FUNCTION_BLOCK FB_MonetTelescopeControl EXTENDS FB_AltAzTelescopeControl IMPLEMENTS I_AltAzTelescope
VAR_INPUT
	fbFocus				: I_Focus;
	fbCovers			: I_MirrorCovers;
	fbBrake				: I_Brake;	
	fbHydraulics   		: I_Hydraulics;
	fbElevation			: REFERENCE TO FB_ElevationControl;
	fbAzimuth			: REFERENCE TO FB_AzimuthControl;
	fbDerotator			: REFERENCE TO FB_DerotatorControl;

	bBrakeClearing		: BOOL	:= TRUE;
END_VAR
VAR_OUTPUT
	fDerotatorSign		: LREAL := 1.0;	// derotator
	
	fElevationPointingOffset : LREAL;
	fAzimuthPointingOffset : LREAL;
	fElevationPointingOffset2 : LREAL;
	fAzimuthPointingOffset2 : LREAL;
	
	fRightAscensionCurrentSky: LREAL;
	fDeclinationCurrentSky: LREAL;

	fDerotatorVelocity	: LREAL;	// rotational velocity of the derotator
	fElevationVelocity	: LREAL;	// rotational velocity of the elevation
	fAzimuthVelocity	: LREAL;	// rotational velocity of the elevation
END_VAR
VAR
	fbPointing			: FB_PointingModelForward(AOFF := 0.0, BNP := 0.0, AN_A := 0.0, AE_A := 0.0, NPAE := 0.0, 
                                                  EOFF := 0.0, AN_E := 0.0, AE_E := 0.0, TF := 0.0);
	fbPointingInverse	: FB_PointingModelInversion(fbPointing := fbPointing);
END_VAR

// get the system time
fbTime();
fJd := DateTime2JD(fbTime.time_RTCEX2);
fLst := CT2LST(telescopeConfig.longitude, fJd);

// set reset state either by hardware (key pressed) or by software (set by e.g. tcs)
rtrigReset(CLK := bReset);

IF bReset THEN
	bHorizonError := FALSE; // if reset, the bHorizonError can be switched off
	
	// reset the stages of all statemachine methods
	bInterrupted := TRUE; 
	_HomeTelescope();
	_GotoTelescope();
	_SlewTelescope();
	_ParkTelescope();
	bInterrupted := FALSE;
END_IF

// get error ID, reset if bReset command is set
IF fbAzimuth.Error THEN
	nErrorID := fbAzimuth.nErrorID;
	IF bReset THEN
		fbAzimuth.Reset();
	END_IF
ELSIF fbElevation.bError THEN
	nErrorID := fbElevation.nErrorID;
	IF bReset THEN
		fbElevation.Reset();
	END_IF
ELSIF fbDerotator.bError THEN
	nErrorID := fbDerotator.nErrorID;
	IF bReset THEN
		fbDerotator.Reset();
	END_IF	
ELSIF fbFocus <> 0 AND_THEN fbFocus.Error THEN
	nErrorID := fbFocus.ErrorID;
	IF bReset THEN
		fbFocus.Reset();
	END_IF
END_IF

// fSlewTime
fSlewTime :=  MAX(MAX(fbElevation.fSlewTime, fbAzimuth.fSlewTime), fbDerotator.fSlewTime);

bError := fbElevation.Error OR 
		 fbAzimuth.bError OR
		 (fbFocus <> 0 AND_THEN fbFocus.Error) OR
		 fbDerotator.bError;
			
IF bError THEN
	bGoHome := 	FALSE;
	bTrack := 	FALSE;
	bGoto := 	FALSE;
	bSlew := 	FALSE;
	fbElevation.Enable := FALSE;
	fbAzimuth.Enable := FALSE;
	fbDerotator.Enable := FALSE;
ELSE
	nErrorID := 0;
END_IF

IF fbElevation.bError THEN
	fbElevation.Enable := FALSE;
	fbAzimuth.Enable := FALSE;
	fbDerotator.Enable := FALSE;
	fbBrake.CloseBrake();
END_IF

eq2hor(
	ra := fRightAscension,
	dec := fDeclination,
	lon := telescopeConfig.longitude,
	lat := telescopeConfig.latitude,
	altitude := telescopeConfig.altitude,
	JD := fJd + fTimeOffset,
	refract_to_observed := TRUE,
	// refract := FALSE,
	alt => fElevationCalc,
	az => fAzimuthCalc,
	ha => fHourAngleCalc);

// apply pointing model
fbPointing(
	fAzimuth			:= fAzimuthCalc,
	fElevation			:= fElevationCalc,
	fAzimuthOffset		=> fAzimuthPointingOffset,
	fElevationOffset	=> fElevationPointingOffset
);
fElevationCalc := fElevationCalc + fElevationPointingOffset + fElevationOffset;
fAzimuthCalc := fAzimuthCalc + fAzimuthPointingOffset + fAzimuthOffset / COS(fElevationCalc * d2r);

// calculate derotator position 
fDerotatorCalc := F_DerotatorPosition2(fAzimuthCalc, fElevationCalc, fDeclination, telescopeConfig.latitude, fDerotatorSign)  + fDerotatorOffset;

// calculate velocities
fDerotatorVelocity := F_Derotatorvelocity(fElevationCalc, fAzimuthCalc, telescopeConfig.latitude);
fElevationVelocity := F_Elevationvelocity(fAzimuthCalc, telescopeConfig.latitude);
fAzimuthVelocity := F_Azimuthvelocity(fElevationCalc, fAzimuthCalc, telescopeConfig.latitude);

// calculate velocities
fDerotatorVelocity := F_Derotatorvelocity(fElevationCalc, fAzimuthCalc, telescopeConfig.latitude);
fElevationVelocity := F_Elevationvelocity(fAzimuthCalc, telescopeConfig.latitude);
fAzimuthVelocity := F_Azimuthvelocity(fElevationCalc, fAzimuthCalc, telescopeConfig.latitude);

IF (fAzimuthCalc > 270.0) THEN
	fAzimuthCalc := fAzimuthCalc - 360.0;
ELSIF (fAzimuthCalc < -274.0) THEN
	fAzimuthCalc := fAzimuthCalc + 360.0;
END_IF
IF (fDerotatorCalc > 360.0) THEN
	fDerotatorCalc := fDerotatorCalc - 360.0;
ELSIF (fDerotatorCalc < -90.0) THEN
	fDerotatorCalc := fDerotatorCalc + 360.0;
END_IF

//IF (fAzimuthCalc > 310.0 AND fAzimuthVelocity > 0.0) OR (fAzimuthCalc > 440.0) THEN
//	fAzimuthCalc := fAzimuthCalc - 360.0;
//ELSIF (fAzimuthCalc < 80.0 AND fAzimuthVelocity < 0.0) OR (fAzimuthCalc < -50.0) THEN
//	fAzimuthCalc := fAzimuthCalc + 360.0;
//END_IF

//IF (fDerotatorCalc > 290.0 AND fDerotatorVelocity > 0.0) OR (fDerotatorCalc > 380.0) THEN
//	fDerotatorCalc := fDerotatorCalc - 360.0;
//ELSIF (fDerotatorCalc < 20.0 AND fDerotatorVelocity < 0.0) OR (fDerotatorCalc < -70.0) THEN
//	fDerotatorCalc := fDerotatorCalc + 360.0;
//END_IF

// get current coordinates	
fAzimuthCurrent := fbAzimuth.fActualPosition;
fElevationCurrent := fbElevation.fActualPosition;
fDerotatorCurrent := fbDerotator.fActualPosition;

// apply inverse pointing model
fbPointingInverse(
	fAzimuth			:= fAzimuthCurrent,
	fElevation			:= fElevationCurrent,
	fAzimuthOffset  	=> fAzimuthPointingOffset2,
	fElevationOffset	=> fElevationPointingOffset2
);
fAzimuthCurrentSky := fAzimuthCurrent - fAzimuthPointingOffset2;
fElevationCurrentSky := fElevationCurrent - fElevationPointingOffset2;

// add offsets
//fElevationCurrent := fElevationCurrentSky - fElevationOffset;
//fAzimuthCurrent := fAzimuthCurrentSky - fAzimuthOffset / COS(fElevationCalc * d2r);

// calculate equatorial coordinates
hor2eq(alt := fElevationCurrentSky - fElevationOffset, 
		az := fAzimuthCurrentSky - fAzimuthOffset / COS(fElevationCalc * d2r),
		jd := fJd,
		lat := telescopeConfig.latitude,
		lon := telescopeConfig.longitude,
		altitude := telescopeConfig.altitude,
		refract_to_observed := FALSE,
		// refract := FALSE,
		ra => fRightAscensionCurrent,
		dec => fDeclinationCurrent);		
hor2eq(alt := fElevationCurrentSky, 
		az := fAzimuthCurrentSky,
		jd := fJd,
		lat := telescopeConfig.latitude,
		lon := telescopeConfig.longitude,
		altitude := telescopeConfig.altitude,
		refract_to_observed := FALSE,
		ra => fRightAscensionCurrentSky,
		dec => fDeclinationCurrentSky);
	
// If the Telescope dips under the fHorizon (e.g. while tracking, stop and gohome)
IF fbElevation.Calibrated AND fElevationCurrent < (fHorizon+0.2) THEN
	IF NOT bStopped AND NOT bGoHome THEN
		bStop := TRUE;
	ELSE
		bGoHome := TRUE;
	END_IF
END_IF
		
tpPowerOnWarning(IN := bPower OR (NOT fbElevation.bEnable AND fbBrake.BrakeOpen), PT := T#250MS);

tonPowerTimeout(IN := TCS_command = E_TCSCommand.no_command AND NOT bIsParked, PT := T#12H);
tonCommandTimeout();
IF tonPowerTimeout.Q AND NOT bIsParked THEN
	bPark := TRUE;
END_IF
		
// set TCS_command according to state variables ordered by precedence
IF bPower THEN
	TCS_command := E_TCSCommand.poweron;
	
ELSIF bStop THEN
	bTrack := FALSE;
	
	// If the stop is during a movement, reset the stage of the movement first
	IF bPark THEN
		bPark := FALSE;
		_ParkTelescope();
	ELSIF bGoto THEN
		bGoto := FALSE;
		_GotoTelescope();
	ELSIF bSlew THEN
		bSlew := FALSE;
		_SlewTelescope();
	ELSIF bGoHome THEN
		bGoHome := FALSE;
		_HomeTelescope();
	END_IF
	TCS_command := E_TCSCommand.stop;
	
ELSIF bPark THEN
	bTrack := FALSE;
	// If lower presedence commands are ongoing, let them know they are interupted
	IF bGoto OR bSlew OR bGoHome THEN
		bGoHome := FALSE;
		bGoto := FALSE;
		bSlew := FALSE;
		bInterrupted := TRUE;
		_HomeTelescope();
		_GotoTelescope();
		_SlewTelescope();
		
	ELSE
		IF bReady AND NOT bBusy THEN
			bInterrupted := FALSE;
			TCS_command := E_TCSCommand.park;
		END_IF
	END_IF
	
ELSIF bGoHome THEN
	bTrack := FALSE;
	// If lower presedence commands are ongoing, let them know they are interupted
	IF bGoto OR bSlew THEN
		bGoto := FALSE;
		bSlew := FALSE;
		bInterrupted := TRUE;
		_GotoTelescope();
		_SlewTelescope();
		
	ELSE
		IF bReady AND NOT bBusy AND bStopped THEN
			bInterrupted := FALSE;
			TCS_command := E_TCSCommand.gohome;
		END_IF
	END_IF
	
	
ELSIF bGoto THEN
	bTrack := FALSE;
	// If lower presedence commands are ongoing, let them know they are interupted
	IF bSlew THEN
		bSlew := FALSE;
		bInterrupted := TRUE;
		_SlewTelescope();
	ELSE
		IF bReady AND NOT bBusy THEN
			bInterrupted := FALSE;
			TCS_command := E_TCSCommand.goto;
		END_IF
	END_IF
		
ELSIF bSlew THEN
	bTrack := FALSE;
	IF bReady AND NOT bBusy THEN
		TCS_command := E_TCSCommand.slew;
	END_IF
	
ELSIF bTrack THEN
	IF bReady AND NOT bBusy THEN
		TCS_command := E_TCSCommand.track;
	END_IF
	
ELSE
	TCS_command := E_TCSCommand.no_command;
	fbElevation.bMoveAxis := FALSE;
	fbAzimuth.bMoveAxis := FALSE;
	fbDerotator.bMoveAxis := FALSE;
	fbElevation.bTracking := FALSE;
	fbAzimuth.bTracking := FALSE;
	fbDerotator.bTracking := FALSE;
END_IF

IF TCS_command = E_TCSCommand.poweron THEN
	_PowerOn();
	tonCommandTimeout(IN := TCS_command = E_TCSCommand.poweron, PT := T#12H);
	TCSCTOEvent.OnMessage := 'POWER';
ELSIF TCS_command = E_TCSCommand.stop THEN
	_StopTelescope();
	tonCommandTimeout(IN := TCS_command = E_TCSCommand.stop, PT := T#2S);
	TCSCTOEvent.OnMessage := 'STOP';
ELSIF TCS_command = E_TCSCommand.park THEN
	_ParkTelescope();
	tonCommandTimeout(IN := TCS_command = E_TCSCommand.park, PT := T#2M);
	TCSCTOEvent.OnMessage := 'PARK';
ELSIF TCS_command = E_TCSCommand.gohome THEN
	_HomeTelescope();
	tonCommandTimeout(IN := TCS_command = E_TCSCommand.gohome, PT := T#2M);
	TCSCTOEvent.OnMessage := 'GOHOME';
ELSIF TCS_command = E_TCSCommand.goto THEN
	_GotoTelescope();
	tonCommandTimeout(IN := TCS_command = E_TCSCommand.goto, PT := T#2M);
	TCSCTOEvent.OnMessage := 'GOTO';
ELSIF TCS_command = E_TCSCommand.slew THEN
	_SlewTelescope();
	tonCommandTimeout(IN := TCS_command = E_TCSCommand.slew, PT := T#2M);
	TCSCTOEvent.OnMessage := 'SLEW';
ELSIF TCS_command = E_TCSCommand.track THEN
	_TrackTelescope();
	tonCommandTimeout(IN := TCS_command = E_TCSCommand.track, PT := T#12H);
	TCSCTOEvent.OnMessage := 'TRACK';
ELSE
	// disable command timeout
	tonCommandTimeout(IN := FALSE);
	TCSCTOEvent.OnMessage := 'NOCOMMAND';
END_IF
 
bSlewing := NOT bTracking AND (fbElevation.fbAxis.InMotion OR fbElevation.fbAxis.InRamp OR
			fbAzimuth.fbAxis.InMotion OR fbAzimuth.fbAxis.InRamp OR
			fbDerotator.fbAxis.InMotion OR fbDerotator.fbAxis.InRamp);

// signal must be stable for 5500MS
tonTrackingDelay(in := fbElevation.fbAxis.isTracking AND 
			fbAzimuth.fbAxis.isTracking AND
			fbDerotator.fbAxis.isTracking,PT :=T#5500MS, Q => bTracking);
			
bStopped :=  (NOT fbElevation.bEnable OR fbElevation.fbAxis.StandStill) AND 
			(NOT fbAzimuth.bEnable OR fbAzimuth.fbAxis.StandStill) AND
			(NOT fbDerotator.bEnable OR fbDerotator.fbAxis.StandStill);
			
bHomed := fbElevation.Calibrated AND
			fbAzimuth.Calibrated AND
			fbFocus.Calibrated AND
			fbDerotator.Calibrated;
			
bReady := bHomed AND 
	fbCovers.Opened AND 
	fbElevation.bEnable AND
	fbAzimuth.bEnable AND
	fbDerotator.bEnable AND fbBrake.BrakeOpen AND 
    NOT bError;

bBusy := fbElevation.fbAxis.Busy OR
		fbAzimuth.fbAxis.Busy OR
		fbDerotator.fbAxis.Busy OR
		fbFocus.Busy;

(* STATUS STATES*)
//fReadyState (see also _PowerOn and _ParkTelescope calls above)
IF bReady THEN
	fReadyState := 1.0;
ELSIF bError THEN
	fReadyState := -1.0;
ELSIF bPower THEN
	fReadyState := 0.7;
ELSIF bIsParked THEN
	fReadyState := 0.0;
ELSIF bPark THEN
	fReadyState := 0.3;
END_IF

//MotionState
IF bStopped THEN
	nMotionState := 0;
ELSIF bSlewing OR bBusy THEN
	nMotionState := 1;
ELSIF bTracking THEN
	nMotionState := 8;
END_IF

// unset the STOP command if telescope is already stopped
IF bStopped THEN
	bStop := FALSE;
END_IF
	
IF NOT bError THEN
	bReset := FALSE;
END_IF

IF bEstopTriggered THEN
	fbElevation.Enable := FALSE;
	fbAzimuth.Enable := FALSE;
	fbDerotator.Enable := FALSE;
END_IF

// send telemetry
IF bSlewing OR bTrack OR bTracking THEN
	tonMQTTTimer.PT := T#500MS; // during movement every second
ELSE
	tonMQTTTimer.PT := T#1000MS; // otherwise every five seconds
END_IF
tonMQTTTimer(IN:=TRUE);
IF tonMQTTTimer.Q THEN
	tonMQTTTimer(IN:=FALSE);
	_SendTelemetry();
END_IF


(* Event function blocks start here. *)
TCSpowerEvent(	Trigger := bPowerFailure, 
				Level := ADSLOG_MSGTYPE_ERROR,
				FormatString := 'power %s',
				//OnMessage := 'Failure',
				OffMessage := 'OK', 
				Comm := fbComm);

TCSgohomeEvent(	Trigger := bGoHome, 
				Level := ADSLOG_MSGTYPE_HINT,
				FormatString := 'GOHOME %s',
				OnMessage := 'commencing',
				OffMEssage := 'completed', 
				Comm := fbComm);
TCSparkEvent(	Trigger := bPark, 
				Level := ADSLOG_MSGTYPE_HINT,
				FormatString := 'PARK %s',
				OnMessage := 'commencing',
				OffMEssage := 'completed', 
				Comm := fbComm);
TCSgotoEvent(	Trigger := bGoto, 
				Level := ADSLOG_MSGTYPE_HINT,
				FormatString := 'GOTO %s',
				OnMessage := 'commencing',
				OffMEssage := 'completed', 
				Comm := fbComm);
TCStrackEvent(	Trigger := bTrack, 
				Level := ADSLOG_MSGTYPE_HINT,
				FormatString := 'TRACK %s',
				OnMessage := 'commencing',
				OffMEssage := 'completed', 
				Comm := fbComm);
TCSstopEvent(	Trigger := bStop, 
				Level := ADSLOG_MSGTYPE_WARN,
				FormatString := 'STOP %s',
				OnMessage := 'commencing',
				OffMEssage := 'completed',
				OffLevel := ADSLOG_MSGTYPE_HINT, 
				Comm := fbComm);
TCStargetHorizonEvent(	Trigger := bPower AND fElevationCalc<fHorizon, 
				Level := ADSLOG_MSGTYPE_WARN,
				FormatString := '%s',
				OnMessage := 'Target below safe horizon',
				OffMEssage := '', 
				Comm := fbComm);
TCSreadyEvent(	Trigger := bPower AND bReady, 
				Level := ADSLOG_MSGTYPE_HINT,
				FormatString := '%s',
				OnMessage := 'STELLA1 startup finished', 
				Comm := fbComm);
TCSCTOEvent(	Trigger := tonCommandTimeout.Q,
				Level := ADSLOG_MSGTYPE_WARN,
				FormatString := 'A timeout occured during %s command!',
				OnMessage := 'NOCOMMAND', 
				Comm := fbComm);

METHOD PRIVATE _GotoTelescope : USINT
VAR_INPUT
END_VAR
VAR
	GoToEvent		: FB_Eventlog;
	commandTimeout	: TON;
END_VAR
VAR_STAT
	nStage			: USINT := 0;
	nLastStage		: USINT := 101;
END_VAR
_GotoTelescope := nStage;
commandTimeout(IN := nStage < 100, PT := T#600S);
IF commandTimeout.Q THEN
	bError := TRUE;
	nErrorID := 16#10;
	bGoto := FALSE;
	nStage := 0;
	RETURN;
END_IF

IF fElevationCalc<2.0 THEN
	bError := TRUE;
	nErrorID := 16#15;
	bGoto := FALSE;
	nStage := 0;
	RETURN;
END_IF

IF bReset OR bError OR bInterrupted THEN
	nStage := 0;
	RETURN;
END_IF

CASE nStage OF
	0:	
		IF bReady AND NOT bBusy THEN
			nStage := 10;
		END_IF
	10:
		IF fbElevation.Tracking = TRUE OR fbAzimuth.Tracking = TRUE OR fbDerotator.Tracking = TRUE THEN
			fbElevation.Tracking := FALSE;
			fbAzimuth.Tracking := FALSE;
			fbDerotator.Tracking := FALSE;
		ELSE
			nStage := 25;
		END_IF				
	25:	
		fbElevation.Position := fElevationCalc;
		fbAzimuth.Position := fAzimuthCalc;
		fbDerotator.Position := fDerotatorCalc;
		fbDerotator.Velocity := 10.0;
		fbElevation.Velocity := 10.0;
		fbAzimuth.Velocity := 10.0;
		
		fbElevation.MoveAxis := TRUE;
		fbAzimuth.MoveAxis := TRUE;
		fbDerotator.MoveAxis := TRUE;
		IF fbElevation.Busy AND
			fbAzimuth.Busy AND
			fbDerotator.Busy THEN
				nStage := 50;
		END_IF
	50:
		IF NOT fbElevation.Busy AND fbElevation.MoveDone THEN
			fbElevation.MoveAxis := FALSE;
		END_IF
		IF NOT fbAzimuth.Busy AND fbAzimuth.MoveDone THEN
			fbAzimuth.MoveAxis := FALSE;
		END_IF
		IF NOT fbDerotator.Busy AND fbDerotator.MoveDone THEN
			fbDerotator.MoveAxis := FALSE;
		END_IF
		IF NOT fbElevation.MoveAxis AND 
           NOT fbAzimuth.MoveAxis AND 
		   NOT fbDerotator.MoveAxis THEN
		   nStage := 75;
		END_IF
	75:
		IF NOT bSlewing AND bStopped THEN // all axis standstill
			nStage := 100;
		END_IF
	100:
		fbElevation.MoveAxis := FALSE;
		fbAzimuth.MoveAxis := FALSE;
		fbDerotator.MoveAxis := FALSE;
		fAzimuth := fAzimuthCalc;
		fElevation := fElevationCalc;
		bGoto := FALSE;
		// enable automatic tracking
		bTrack := bAutoTrack;
		nStage := 0;
END_CASE
GoToEvent(Trigger := nStage > nLastStage, FormatString := 'GoTo progress: %s', OnMessage := USINT_TO_STRING(nStage), comm := fbComm);
nLastStage := nStage;
END_METHOD

METHOD PRIVATE _HomeTelescope : BOOL
VAR_INPUT
END_VAR
VAR
	HomeEvent		: FB_Eventlog;
	commandTimeout	: TON;
END_VAR
commandTimeout(IN := NOT _HomeTelescope, PT := T#600S);
IF commandTimeout.Q THEN
	bError := TRUE;
	nErrorID := 16#30;
	_HomeTelescope :=TRUE;
END_IF

IF bReady AND bStopped AND NOT bBusy AND NOT bTracking THEN
	fbElevation.Velocity := 10.0;
	fbElevation.Position := telescopeConfig.elevationHome;
	fbElevation.MoveAxis := TRUE;
	fbAzimuth.Velocity := 10.0;
	fbAzimuth.Position := telescopeConfig.azimuthHome;
	fbAzimuth.MoveAxis := TRUE;
	fbDerotator.Velocity := 10.0;
	fbDerotator.Position := telescopeConfig.derotatorHome;
	fbDerotator.MoveAxis := TRUE;	
END_IF

IF fbElevation.MoveDone AND 
	fbAzimuth.MoveDone AND 
	fbDerotator.MoveDone THEN
	bGoHome := FALSE;
	fElevation := fElevationCurrent;
	fAzimuth := fAzimuthCurrent;
	_HomeTelescope := TRUE;
ELSE
	_HomeTelescope := FALSE;
END_IF

HomeEvent(Trigger := _HomeTelescope, 
			Level := ADSLOG_MSGTYPE_HINT,
			FormatString := '%s',
			OnMessage := 'Telescope is homed.', comm := fbComm);
END_METHOD

METHOD PRIVATE _ParkTelescope : USINT
VAR_INPUT
END_VAR
VAR
	ParkEvent	: FB_Eventlog;
END_VAR
VAR_STAT
	nStage		: USINT := 0;
	nLastStage	: USINT := 101;
END_VAR
_ParkTelescope := nStage;
IF bReset OR bError OR bStop OR bInterrupted THEN
	nStage := 0;
	RETURN;
END_IF
IF bIsParked THEN
	nStage := 100;
END_IF
CASE nStage OF
	0: 
		bGoHome := 	FALSE;
		bTrack := 	FALSE;
		bGoto := 	FALSE;
		bSlew := 	FALSE;
		IF fbFocus <> 0 THEN
			fbFocus.Position := telescopeConfig.focusPark;
		END_IF
		IF bError THEN // emergency park
			fbBrake.CloseBrake();
			fbElevation.Enable := FALSE;
			fbAzimuth.Enable := FALSE;
			fbDerotator.Enable := FALSE;	
			fbCovers.Close();	
			nStage := 80;
		END_IF
		nStage := 10;
	10:
		IF fbElevation.Tracking = TRUE OR fbAzimuth.Tracking = TRUE OR fbDerotator.Tracking = TRUE THEN
			fbElevation.Tracking := FALSE;
			fbAzimuth.Tracking := FALSE;
			fbDerotator.Tracking := FALSE;
		ELSE
			nStage := 20;
		END_IF		
	20:
		fbElevation.Position := telescopeConfig.elevationPark;
		fbElevation.Velocity := 10.0;
		fbElevation.MoveAxis := TRUE;
		fbAzimuth.Position := telescopeConfig.azimuthPark;
		fbAzimuth.Velocity := 10;
		fbAzimuth.MoveAxis := TRUE;
		fbDerotator.Position := telescopeConfig.derotatorPark;
		fbDerotator.Velocity := 10.0;
		fbDerotator.MoveAxis := TRUE;
		IF fbElevation.Busy AND
			fbAzimuth.Busy AND
			fbDerotator.Busy THEN
				nStage := 40;
		END_IF
	40:
		IF fbElevation.MoveDone THEN
			fbElevation.MoveAxis := FALSE;
		END_IF
		IF fbAzimuth.MoveDone THEN
			fbAzimuth.MoveAxis := FALSE;
		END_IF
		IF fbDerotator.MoveDone THEN
			fbDerotator.MoveAxis := FALSE;
		END_IF
		IF NOT bSlewing THEN // all axis standstill
			nStage := 60;
		END_IF
	60:
		IF NOT fbElevation.Enable AND NOT fbAzimuth.Enable AND NOT fbDerotator.Enable THEN
			nStage := 80;
		END_IF

		IF bStopped THEN
			fbElevation.Enable := FALSE;
			fbAzimuth.Enable := FALSE;
			fbDerotator.Enable := FALSE;
		END_IF
		
		fbElevation.bMoveAxis := FALSE;
		fbAzimuth.bMoveAxis := FALSE;
		fbDerotator.bMoveAxis := FALSE;
	80:
		IF fbElevation.Enable OR fbAzimuth.Enable OR fbDerotator.Enable THEN
			nStage := 60;
		END_IF
		IF NOT fbBrake.BrakeOpen THEN
			fbCovers.Close();
			fbHydraulics.Enable := FALSE;
		END_IF
		IF fbCovers.Closed THEN
			nStage := 100;
		END_IF
	100:
			bIsParked := TRUE;
			bPark := FALSE;
			_ParkTelescope := 100;
			nStage := 0;	
END_CASE
ParkEvent(Trigger := nStage > nLastStage, FormatString := 'Parking progress: %s', OnMessage := USINT_TO_STRING(nStage), comm := fbComm);
nLastStage := nStage;
END_METHOD

METHOD PRIVATE _PowerOn : BOOL
VAR_INPUT
END_VAR
IF NOT bBrakeClearing THEN
	bPowerFailure := TRUE;
	TCSpowerEvent.OnMessage := 'failure: brake clearing not set';
	bPower := FALSE;
ELSIF bError THEN
	bPowerFailure := TRUE;
	TCSpowerEvent.OnMessage := 'Generic error during power on occured.';
	bPower := FALSE;
ELSE
	bPowerFailure := FALSE;		
END_IF
// COVER MUST BE OPENED FOR A SUCCESSFUL WAKE & SHAKE COMMAND!
fbCovers.Open();

// enable elevation, enable azimuth
IF bMainReady AND fbCovers.Opened THEN
	fbElevation.Enable := TRUE;
	fbAzimuth.Enable := TRUE;
	fbDerotator.Enable := TRUE;
END_IF

IF fbElevation.Ready AND NOT fbElevation.Calibrated THEN
	fbElevation.HomeAxis := TRUE;
END_IF

IF fbAzimuth.Ready AND NOT fbAzimuth.Calibrated THEN
	fbAzimuth.HomeAxis := TRUE;
END_IF

// enable derotator
IF fbElevation.Ready THEN
	fbDerotator.HomeAxis := fbDerotator.Ready AND NOT fbDerotator.Calibrated;
END_IF

// start calibration of focus after elevation has been calibrated
// this avoids imbalance by the M2 mirror on the elvation during its calibration
IF fbElevation.Calibrated AND (fbFocus <> 0 AND_THEN NOT fbFocus.Calibrated) THEN
	fbFocus.Enable := TRUE;
	fbFocus.HomeAxis := TRUE;
END_IF

IF fbCovers.Opened AND 
	fbElevation.Calibrated AND
	fbAzimuth.Calibrated AND
	fbDerotator.Calibrated THEN
	//FocusControl.Calibrated THEN
	bPower := FALSE;
	_PowerOn := TRUE;
	bIsParked := FALSE;
	// slew the telescope to the home position
	bGoHome := TRUE;
ELSE
	_PowerOn := FALSE;
END_IF
END_METHOD

METHOD _SendTelemetry : BOOL
VAR_INPUT
END_VAR
SUPER^._PublishTelemetry();

fbComm.Publish('telescope', 'dome', 'TELESCOPE.READY_STATE',	LREAL_TO_STRING(fReadyState));
fbComm.Publish('telescope', 'dome', 'TELESCOPE.MOTION_STATE',	LREAL_TO_STRING(nMotionState));

// INFO
fbComm.Publish('telescope', 'dome', 'TELESCOPE.INFO.NAME',	telescopeConfig.name);
fbComm.Publish('telescope', 'dome', 'TELESCOPE.INFO.DIAMETER',	LREAL_TO_STRING(telescopeConfig.diameter));
fbComm.Publish('telescope', 'dome', 'TELESCOPE.INFO.CABINET',	telescopeConfig.cabinet);
fbComm.Publish('telescope', 'dome', 'TELESCOPE.INFO.MANUFACTURER', telescopeConfig.manufacturer);

// config
fbComm.Publish('telescope', 'dome', 'TELESCOPE.CONFIG.MOUNTOPTIONS', telescopeConfig.mountOptions);
fbComm.Publish('telescope', 'dome', 'TELESCOPE.CONFIG.MOUNT', telescopeConfig.mount);

// STATUS
IF bEstopTriggered THEN
	fbComm.Publish('telescope', 'dome', 'TELESCOPE.STATUS.GLOBAL', '1');
ELSIF bError THEN
	fbComm.Publish('telescope', 'dome', 'TELESCOPE.STATUS.GLOBAL', '2');
ELSE
	fbComm.Publish('telescope', 'dome', 'TELESCOPE.STATUS.GLOBAL', '0');
END_IF

// INSTRUMENTAL
fbComm.Publish('telescope', 'dome', 'OBJECT.INSTRUMENTAL.ALT', LREAL_TO_STRING(fElevation));
fbComm.Publish('telescope', 'dome', 'OBJECT.INSTRUMENTAL.AZ', LREAL_TO_STRING(fAzimuth));

// EQUATORIAL
fbComm.Publish('telescope', 'dome', 'OBJECT.EQUATORIAL.EPOCH', 'J2000.0');
fbComm.Publish('telescope', 'dome', 'OBJECT.EQUATORIAL.EQUINOX', 'J2000.0');
fbComm.Publish('telescope', 'dome', 'OBJECT.EQUATORIAL.RA_PM', '0.0');
fbComm.Publish('telescope', 'dome', 'OBJECT.EQUATORIAL.DEC_PM', '0.0');
fbComm.Publish('telescope', 'dome', 'OBJECT.EQUATORIAL.RA_RATE', '0.0');
fbComm.Publish('telescope', 'dome', 'OBJECT.EQUATORIAL.DEC_RATE', '0.0');
fbComm.Publish('telescope', 'dome', 'OBJECT.EQUATORIAL.RA', LREAL_TO_STRING(fRightAscension/15.0));
fbComm.Publish('telescope', 'dome', 'OBJECT.EQUATORIAL.DEC', LREAL_TO_STRING(fDeclination));	

// HORIZONTAL
fbComm.Publish('telescope', 'dome', 'OBJECT.HORIZONTAL.ALT', LREAL_TO_STRING(fElevationCalc));
fbComm.Publish('telescope', 'dome', 'OBJECT.HORIZONTAL.AZ', LREAL_TO_STRING(fAzimuthCalc));

(* POINTING *)
fbComm.Publish('telescope', 'dome', 'POINTING.SLEWTIME', LREAL_TO_STRING(fSlewtime));
fbComm.Publish('telescope', 'dome', 'POINTING.OFFSETS.ALT', LREAL_TO_STRING(fElevationPointingOffset));
fbComm.Publish('telescope', 'dome', 'POINTING.OFFSETS.AZ', LREAL_TO_STRING(fAzimuthPointingOffset));

(*POSITION*)
//LOCAL
fbComm.Publish('telescope', 'dome', 'POSITION.LOCAL.SIDEREAL_TIME', LREAL_TO_STRING(fLst));
fbComm.Publish('telescope', 'dome', 'POSITION.LOCAL.JD', LREAL_TO_STRING(fJd));
fbComm.Publish('telescope', 'dome', 'POSITION.LOCAL.LATITUDE', LREAL_TO_STRING(telescopeConfig.latitude));
fbComm.Publish('telescope', 'dome', 'POSITION.LOCAL.LONGITUDE', LREAL_TO_STRING(telescopeConfig.longitude));
fbComm.Publish('telescope', 'dome', 'POSITION.LOCAL.HEIGHT', LREAL_TO_STRING(telescopeConfig.altitude));

// INSTRUMENTAL
// > ALT
// POWER_STATE
IF fbElevation.Enable THEN
	fbComm.Publish('telescope', 'dome', 'POSITION.INSTRUMENTAL.ALT.POWER_STATE', '1.0');
ELSE
	fbComm.Publish('telescope', 'dome', 'POSITION.INSTRUMENTAL.ALT.POWER_STATE', '0.0');
END_IF
//REFERENCED
IF fbElevation.Calibrated THEN
	fbComm.Publish('telescope', 'dome', 'POSITION.INSTRUMENTAL.ALT.REFERENCED', '1.0');
ELSE
	fbComm.Publish('telescope', 'dome', 'POSITION.INSTRUMENTAL.ALT.REFERENCED', '0.0');
END_IF
//ERROR_STATE
IF fbElevation.Error THEN
	fbComm.Publish('telescope', 'dome', 'POSITION.INSTRUMENTAL.ALT.ERROR_STATE', UDINT_TO_STRING(fbElevation.ErrorID));
ELSE
	fbComm.Publish('telescope', 'dome', 'POSITION.INSTRUMENTAL.ALT.ERROR_STATE', '0');
END_IF
//MOTION_STATE
IF fbElevation.Busy THEN
	IF fbElevation.isTracking THEN
		fbComm.Publish('telescope', 'dome', 'POSITION.INSTRUMENTAL.ALT.MOTION_STATE', '8');
	ELSE
		fbComm.Publish('telescope', 'dome', 'POSITION.INSTRUMENTAL.ALT.MOTION_STATE', '1');
	END_IF
ELSE
	fbComm.Publish('telescope', 'dome', 'POSITION.INSTRUMENTAL.ALT.MOTION_STATE', '0');
END_IF
fbComm.Publish('telescope', 'dome', 'POSITION.INSTRUMENTAL.ALT.REALPOS', LREAL_TO_STRING(fElevationCurrent-fElevationOffset));
fbComm.Publish('telescope', 'dome', 'POSITION.INSTRUMENTAL.ALT.CURRPOS', LREAL_TO_STRING(fElevationCurrent));
fbComm.Publish('telescope', 'dome', 'POSITION.INSTRUMENTAL.ALT.TARGETPOS', LREAL_TO_STRING(fbElevation.Position));
fbComm.Publish('telescope', 'dome', 'POSITION.INSTRUMENTAL.ALT.CURRSPEED', LREAL_TO_STRING(fbElevation.Velocity));
fbComm.Publish('telescope', 'dome', 'POSITION.INSTRUMENTAL.ALT.TARGETDISTANCE', LREAL_TO_STRING(ABS(fElevationCurrent-fbElevation.Position)));
fbComm.Publish('telescope', 'dome', 'POSITION.INSTRUMENTAL.ALT.OFFSET', LREAL_TO_STRING(fElevationOffset));

// > AZ
// POWER_STATE
IF fbAzimuth.Enable THEN
	fbComm.Publish('telescope', 'dome', 'POSITION.INSTRUMENTAL.AZ.POWER_STATE', '1.0');
ELSE
	fbComm.Publish('telescope', 'dome', 'POSITION.INSTRUMENTAL.AZ.POWER_STATE', '0.0');
END_IF
//REFERENCED
IF fbAzimuth.Calibrated THEN
	fbComm.Publish('telescope', 'dome', 'POSITION.INSTRUMENTAL.AZ.REFERENCED', '1.0');
ELSE
	fbComm.Publish('telescope', 'dome', 'POSITION.INSTRUMENTAL.AZ.REFERENCED', '0.0');
END_IF
//ERROR_STATE
IF fbAzimuth.Error THEN
	fbComm.Publish('telescope', 'dome', 'POSITION.INSTRUMENTAL.AZ.ERROR_STATE', UDINT_TO_STRING(fbAzimuth.ErrorID));
ELSE
	fbComm.Publish('telescope', 'dome', 'POSITION.INSTRUMENTAL.AZ.ERROR_STATE', '0');
END_IF
//MOTION_STATE
IF fbAzimuth.Busy THEN
	IF fbAzimuth.isTracking THEN
		fbComm.Publish('telescope', 'dome', 'POSITION.INSTRUMENTAL.AZ.MOTION_STATE', '8');
	ELSE
		fbComm.Publish('telescope', 'dome', 'POSITION.INSTRUMENTAL.AZ.MOTION_STATE', '1');
	END_IF
ELSE
	fbComm.Publish('telescope', 'dome', 'POSITION.INSTRUMENTAL.AZ.MOTION_STATE', '0');
END_IF

fbComm.Publish('telescope', 'dome', 'POSITION.INSTRUMENTAL.AZ.CURRPOS', LREAL_TO_STRING(fAzimuthCurrent));
fbComm.Publish('telescope', 'dome', 'POSITION.INSTRUMENTAL.AZ.REALPOS', LREAL_TO_STRING(fAzimuthCurrent-fAzimuthOffset/COS(fElevation*d2r)));
fbComm.Publish('telescope', 'dome', 'POSITION.INSTRUMENTAL.AZ.TARGETPOS', LREAL_TO_STRING(fbAzimuth.Position));
fbComm.Publish('telescope', 'dome', 'POSITION.INSTRUMENTAL.AZ.CURRSPEED', LREAL_TO_STRING(fbAzimuth.Velocity));
fbComm.Publish('telescope', 'dome', 'POSITION.INSTRUMENTAL.AZ.TARGETDISTANCE', LREAL_TO_STRING(ABS(fAzimuthCurrent-fbAzimuth.Position)));
fbComm.Publish('telescope', 'dome', 'POSITION.INSTRUMENTAL.AZ.OFFSET', LREAL_TO_STRING(fAzimuthOffset));


(*HORIZONTAL*)
fbComm.Publish('telescope', 'dome', 'POSITION.HORIZONTAL.ALT', LREAL_TO_STRING(fElevationCurrentSky));
fbComm.Publish('telescope', 'dome', 'POSITION.HORIZONTAL.AZ', LREAL_TO_STRING(fAzimuthCurrentSky));
//fbComm.Publish('telescope', 'dome', 'POSITION.HORIZONTAL.DOME', LREAL_TO_STRING(fbDome.Position));

(*EQUITORIAL*)
fbComm.Publish('telescope', 'dome', 'POSITION.EQUATORIAL.RA_J2000', LREAL_TO_STRING(fRightAscensionCurrent/15.0));
fbComm.Publish('telescope', 'dome', 'POSITION.EQUATORIAL.HA_J2000', LREAL_TO_STRING(fHourAngleCurrent));
fbComm.Publish('telescope', 'dome', 'POSITION.EQUATORIAL.DEC_J2000', LREAL_TO_STRING(fDeclinationCurrent));
END_METHOD

METHOD PRIVATE _SlewTelescope : USINT
VAR_INPUT
END_VAR
VAR
	SlewEvent:	FB_Eventlog;
	command_timeout: TON;
END_VAR
VAR_STAT
	nStage:		USINT := 0;
	nLastStage:	USINT := 101;
END_VAR
_SlewTelescope := nStage;
command_timeout(IN := nStage < 100, PT := T#600S);
IF command_timeout.Q THEN
	bError := TRUE;
	nErrorID := 16#40;
	bSlew := FALSE;
	nStage := 0;
END_IF
IF bReset OR bError OR bInterrupted THEN
	nStage := 0;
END_IF
CASE nStage OF
	0:	
		IF bReady AND bStopped AND NOT bBusy AND NOT bTracking THEN
			nStage := 10;
		END_IF
	10:
		IF fbElevation.Tracking = TRUE OR fbAzimuth.Tracking = TRUE OR fbDerotator.Tracking = TRUE THEN
			fbElevation.Tracking := FALSE;
			fbAzimuth.Tracking := FALSE;
			fbDerotator.Tracking := FALSE;
		ELSE
			nStage := 25;
		END_IF				
	25:
		fbPointing(
			fAzimuth			:= fAzimuth,
			fElevation			:= fElevation,
			fAzimuthOffset		=> fAzimuthPointingOffset,
			fElevationOffset	=> fElevationPointingOffset
		);	
		fbElevation.Position := fElevation + fElevationPointingOffset + fElevationOffset;
		fbElevation.Velocity := 10.0;
		fbElevation.MoveAxis := TRUE;
		fbAzimuth.Position := fAzimuth + fAzimuthPointingOffset + fAzimuthOffset / COS(fElevationCalc * d2r);
		fbAzimuth.Velocity := 10.0;
		fbAzimuth.MoveAxis := TRUE;
		fbDerotator.Position := fElevation + fDerotatorOffset;
		fbDerotator.Velocity := 10.0;
		fbDerotator.MoveAxis := TRUE;
		IF fbElevation.Busy AND
			fbAzimuth.Busy AND
			fbDerotator.Busy THEN
				nStage := 50;
		END_IF
	50:
		IF fbElevation.MoveDone THEN
			fbElevation.bMoveAxis := FALSE;
		END_IF
		
		IF fbAzimuth.MoveDone THEN
			fbAzimuth.MoveAxis := FALSE;
		END_IF

		IF fbDerotator.MoveDone THEN
			fbDerotator.MoveAxis := FALSE;
		END_IF
		IF NOT bSlewing AND bStopped THEN // all axis standstill
			nStage := 100;
		END_IF
	100:
		fbElevation.MoveAxis := FALSE;
		fbAzimuth.MoveAxis := FALSE;
		fbDerotator.MoveAxis := FALSE;
		fRightAscension := fRightAscensionCalc;
		fDeclination := fDeclinationCalc;
		bSlew := FALSE;
		nStage := 0;
END_CASE
SlewEvent(Trigger := nStage > nLastStage, FormatString := 'Slew progress: %s', OnMessage := USINT_TO_STRING(nStage), Comm := fbComm);
nLastStage := nStage;
END_METHOD

METHOD PRIVATE _StopTelescope : BOOL
VAR_INPUT
END_VAR
IF fbAzimuth.Tracking = TRUE OR fbElevation.Tracking = TRUE OR fbDerotator.Tracking = TRUE THEN
	fbAzimuth.Tracking := FALSE;
	fbElevation.Tracking := FALSE;
	fbDerotator.Tracking := FALSE;
ELSIF fbAzimuth.MoveAxis = TRUE OR  fbElevation.MoveAxis = TRUE OR fbDerotator.MoveAxis = TRUE THEN
	fbAzimuth.MoveAxis := FALSE;
	fbElevation.MoveAxis := FALSE;
	fbDerotator.MoveAxis := FALSE;
ELSE
	// Only issue Axis stop commands if they are moving
	IF NOT fbAzimuth.fbAxis.StandStill THEN
		fbAzimuth.StopAxis := TRUE;
	ELSE
		fbAzimuth.StopAxis := FALSE;
	END_IF
	
	IF NOT fbElevation.fbAxis.StandStill THEN
		fbElevation.StopAxis := TRUE;
	ELSE
		fbElevation.StopAxis := FALSE;
	END_IF	
	
	IF NOT fbDerotator.fbAxis.StandStill THEN
		fbDerotator.StopAxis := TRUE;
	ELSE
		fbDerotator.StopAxis := FALSE;
	END_IF	

	IF bStopped THEN
		fbAzimuth.StopAxis := FALSE;
		fbElevation.StopAxis := FALSE;
		fbDerotator.StopAxis := FALSE;
		_StopTelescope := FALSE;
	END_IF
END_IF
END_METHOD

METHOD PRIVATE _TrackTelescope : BOOL
VAR_INPUT
END_VAR
// Elevation
fDerotatorVelocity := F_Derotatorvelocity(fElevationCalc, fAzimuthCalc, telescopeConfig.latitude);
fElevationVelocity := F_Elevationvelocity(fAzimuthCalc, telescopeConfig.latitude);
fAzimuthVelocity := F_Azimuthvelocity(fElevationCalc, fAzimuthCalc, telescopeConfig.latitude);
IF fElevationCurrent < 5.0 OR fElevationCurrent > 89.5 THEN 
	bTrack := FALSE;
END_IF
IF fAzimuthCurrent > 440.0 THEN
	bTrack := FALSE;
END_IF
IF (fDerotatorCurrent < -69.0 AND fDerotatorVelocity<0.0) OR (fDerotatorCurrent > 379.0 AND fDerotatorVelocity>0.0) THEN
	bTrack := FALSE;
END_IF

fbElevation.Position := fElevationCalc;
IF NOT fbElevation.Tracking THEN
	fbElevation.Velocity := 10.0;
	fbElevation.MoveAxis := TRUE;
	IF NOT fbElevation.Busy AND fbElevation.MoveDone THEN
		fbElevation.MoveAxis := FALSE;
		IF fbElevation.isTracking THEN
			fbElevation.Velocity := fElevationVelocity;
		ELSE
			fbElevation.Velocity := 3.0*fElevationVelocity;
		END_IF
		fbElevation.Velocity := fElevationVelocity;
		fbElevation.Tracking := TRUE;
	END_IF
ELSE
	fbElevation.Velocity := fElevationVelocity;
END_IF

// Azimuth
fbAzimuth.Position := fAzimuthCalc;
IF NOT fbAzimuth.Tracking THEN
	fbAzimuth.Velocity := 10.0;
	fbAzimuth.MoveAxis := TRUE;
	IF NOT fbAzimuth.Busy AND fbAzimuth.MoveDone THEN
		fbAzimuth.MoveAxis := FALSE;
		IF fbAzimuth.isTracking THEN
			fbAzimuth.Velocity := fAzimuthVelocity;
		ELSE
			fbAzimuth.Velocity := 3.0*fAzimuthVelocity;
		END_IF
		fbAzimuth.Velocity := fAzimuthVelocity;
		fbAzimuth.Tracking := TRUE;
	END_IF
ELSE
	fbAzimuth.Velocity := fAzimuthVelocity;
END_IF

// Derotator
fbDerotator.Position := fDerotatorCalc;
IF NOT fbDerotator.Tracking THEN
	fbDerotator.Velocity := 10.0;
	fbDerotator.MoveAxis := TRUE;
	IF NOT fbDerotator.Busy AND fbDerotator.MoveDone THEN
		fbDerotator.MoveAxis := FALSE;
		IF fbDerotator.isTracking THEN
			fbDerotator.Velocity := fDerotatorVelocity;
		ELSE
			fbDerotator.Velocity := 3.0*fDerotatorVelocity;
		END_IF
		fbDerotator.Velocity := fDerotatorVelocity;
		fbDerotator.Tracking := TRUE;
	END_IF
ELSE
	fbDerotator.Velocity := fDerotatorVelocity;
END_IF
END_METHOD

{warning 'add property implementation'}
PROPERTY Altitude : LREAL
GET
Altitude := THIS^.fElevationCurrent;
END_GET
END_PROPERTY

{warning 'add property implementation'}
PROPERTY Azimuth : LREAL
GET
Azimuth := THIS^.fAzimuthCurrent;
END_GET
END_PROPERTY

{warning 'add property implementation'}
PROPERTY Declination : LREAL
GET
Declination := THIS^.fDeclination;
END_GET
END_PROPERTY

METHOD Home : BOOL
bGoHome := TRUE;
END_METHOD

METHOD Init : BOOL
bPower := TRUE;
END_METHOD

METHOD MoveAltAz : BOOL
VAR_INPUT
	AltAz	: BROTLib.ST_AltAzCoordinate;
END_VAR
fElevation 	:= AltAz.Altitude;
fAzimuth 	:= AltAz.Azimuth;
bSlew		:= TRUE;
END_METHOD

METHOD MoveRaDec : BOOL
VAR_INPUT
	RaDec	: BROTLib.ST_RaDecCoordinate;
END_VAR
fRightAscension	:= RaDec.RightAscension;
fDeclination	:= RaDec.Declination;
bGoto			:= TRUE;
END_METHOD

METHOD Park : BOOL
bPark := TRUE;
END_METHOD

METHOD Reset : BOOL
bReset := TRUE;
END_METHOD

{warning 'add property implementation'}
PROPERTY RightAscension : LREAL
GET
RightAscension := THIS^.fRightAscension;
END_GET
END_PROPERTY

METHOD SetAltitudeOffset : BOOL
VAR_INPUT
	Offset	: LREAL;
END_VAR
fElevationOffset := Offset;
END_METHOD

METHOD SetAzimuthOffset : BOOL
VAR_INPUT
	Offset	: LREAL;
END_VAR
fAzimuthOffset := Offset;
END_METHOD

METHOD SetDerotatorOffset : BOOL
VAR_INPUT
	Offset	: LREAL;
END_VAR
fDerotatorOffset := Offset;
END_METHOD

{warning 'add method implementation '}
METHOD Slew : BOOL
VAR_INPUT
	fAzimuth	: LREAL;
	fAltitude	: LREAL;
END_VAR
THIS^.fElevation 	:= fAltitude;
THIS^.fAzimuth 	:= fAzimuth;
THIS^.bSlew		:= TRUE;
END_METHOD

METHOD Stop : BOOL
bStop := TRUE;
END_METHOD

{warning 'add method implementation '}
METHOD Track : BOOL
VAR_INPUT
	fRightAscension	: LREAL;
	fDeclination	: LREAL;
END_VAR
THIS^.fRightAscension	:= fRightAscension;
THIS^.fDeclination		:= fDeclination;
//THIS^.bTrack			:= TRUE;
THIS^.bGoto				:= TRUE;
END_METHOD

METHOD TrackRaDec : BOOL
VAR_INPUT
	RaDec	: BROTLib.ST_RaDecCoordinate;
END_VAR
fRightAscension	:= RaDec.RightAscension;
fDeclination		:= RaDec.Declination;
//bTrack			:= TRUE;
THIS^.bGoto				:= TRUE;
END_METHOD

END_FUNCTION_BLOCK

(* stored: Version 1.1.0.1, ProductVersion 3.1.4024.15
   POU FB_MonetTelescopeControl: Id {392c90d3-a441-4c8d-a752-42b25b49f5cd}, SpecialFunc None
   Folder internal methods: Id {d1e7fbc6-9662-4c16-bf25-8044ef92da3b}
   Method _GotoTelescope: Id {8976ce61-8856-40e1-8cfb-7b9454a4edbf}
   Method _HomeTelescope: Id {4753aff7-faba-4306-9d47-8cb63c25adcc}
   Method _ParkTelescope: Id {999576b1-8aca-41eb-91ab-673a6fc7f4ba}
   Method _PowerOn: Id {4c40649f-56d9-4130-9f80-925439540d98}
   Method _SendTelemetry: Id {5e3ab35e-5dd6-4108-99df-8d99cebae004}
   Method _SlewTelescope: Id {d3e1cb80-5564-4d5b-b2d9-2c8dd1b9215a}
   Method _StopTelescope: Id {cb5cd062-03c6-4c9b-bbde-9c71b10960c3}
   Method _TrackTelescope: Id {6e849cc7-222d-486c-8d3d-ea253bc6d574}
   Property Altitude: Id {51b1ff05-1140-4331-8485-239187f5f8b1}
   Get Get: Id {05a6ac86-f3fe-4579-ad82-04708fa0864e}
   Property Azimuth: Id {0dd05217-329b-419a-a3b6-a7f2c3a7b182}
   Get Get: Id {fd6f0d71-0c53-4de5-af62-a6f082f3b2fe}
   Property Declination: Id {b1285964-102f-45b7-af05-6785154ef40d}
   Get Get: Id {add754b0-d14d-4a0e-b482-234fdfd51176}
   Method Home: Id {5b365a4e-cda4-42b8-9d62-ce493e72979f}
   Method Init: Id {78ec73c4-02ac-4d83-aefd-694e0077d330}
   Method MoveAltAz: Id {94f5e9d8-f8f7-4c16-ac3f-2e854a5b373b}
   Method MoveRaDec: Id {86c89766-d350-4f6b-9fea-e302f9b4e7d4}
   Method Park: Id {21fb237d-ad50-4f82-97cf-a56a9c25b954}
   Method Reset: Id {efa0c84e-7359-43c3-a635-1faede103859}
   Property RightAscension: Id {11e4e9e9-9e18-4d9f-ab19-1c208929d2bc}
   Get Get: Id {b17aa26c-317b-4e3f-8426-b76a55e02df1}
   Method SetAltitudeOffset: Id {522d462f-4678-4f02-8df4-00f463761b00}
   Method SetAzimuthOffset: Id {16e0d010-c333-4c19-862e-702e715c040b}
   Method SetDerotatorOffset: Id {f59933b1-4aa9-4f18-88cf-26244adda0df}
   Method Slew: Id {ee4e9e45-2bba-488b-8094-f2bf4a28ec2b}
   Method Stop: Id {d33b3161-dc8a-45e5-ae2f-544550162c16}
   Method Track: Id {36f6a798-1a7b-442f-88f7-fc8d7dfa3dc0}
   Method TrackRaDec: Id {f497d99f-36a3-42c8-ae9b-738903f3158c} *)
